{region '#Template'}
	{attribute 'Version' := '6.0.0.0'}
	{attribute 'Tags' := '"LCID": "1031", "Text": "AC, Aggregates, pre-heater"'}
	{attribute 'Tags' := '"LCID": "1033", "Text": "AC, Aggregates, pre-heater"'}
	{attribute 'Using' := '"Type": "Template", "URI": "Priority"'}		 
	{attribute 'Using' := '"Type": "Template", "URI": "BA2_Param"'}
	{attribute 'Using' := '"Type": "Template", "URI": "EC_ID"'}
	{attribute 'Description' := '"LCID": "1031", "Text": "Aggregat Vorerhitzer"'}
	{attribute 'Description' := '"LCID": "1033", "Text": "Aggregate pre-heater"'}
{endregion}
FUNCTION_BLOCK FB_BA_AC_PreHtr EXTENDS FB_BA_View
VAR_INPUT
	fSpTSuA					: REAL;
	fTSuA					: REAL;
	bSyncTSuACtrl			: BOOL;
	fSyncTSuACtrl			: REAL;	
	bDehumf					: BOOL;
	bSkipPreRinse			: BOOL; // Vorspülen überspringen // Skip pre-rinse
	fTWth					: REAL;
	bTWthLowLimit			: BOOL;
	bResetDehumf    		: BOOL;
END_VAR
VAR_OUTPUT
	bCmd					: BOOL;
	fPresentValue			: REAL;			
	bFrost					: BOOL;
	bPreRinseReady			: BOOL;  
	bActiveSeqCtrl			: BOOL;	
END_VAR
VAR_IN_OUT
	stTSeqLink				: ST_BA_SeqLink; // Sequenz Link Struktur // Sequence link structure	
	stAggregate				: ST_BA_Aggregate;	
END_VAR
VAR_INPUT CONSTANT PERSISTENT
	{attribute 'parameterCategory' := 'Behaviour'}
	fHysPuOn : REAL := 5.0;
	{attribute 'parameterCategory' := 'Behaviour'}
	fHysPuOff : REAL := 1.0;
END_VAR
VAR_INPUT CONSTANT
	TFl						: FB_BA_SensorAnalog;												
	TRt						: FB_BA_SensorAnalog;			
	TSuACtrl				: FB_BA_AC_PreHtrTSuACtrl;
	TRtCtrl					: FB_BA_AC_TRtCtrl;	
	TFrost					: FB_BA_SensorAnalog;																	
	TFrostPrtcCtrlAir		: FB_BA_PID_Sp;
	FrostThermostat			: FB_BA_SensorBinary;
	Vlv						: FB_BA_Vlv;
	Pu						: FB_BA_Pu1st;
	PlantLock				: FB_BA_PlantLock;			
	Aggregate				: FB_BA_Aggregate;																											 							
END_VAR
VAR
	bPrioSfty				: BOOL;
	bPrioCrit				: BOOL;		
	PrioSwiVal				: FB_BA_PrioSwi_B04;	
	
	HysPu					: FB_BA_Swi2P;
	SyncTSuACtrl			: FB_BA_RFTrig;
	SyncSeqCtrlIsActive		: FB_BA_RFTrig;
	PrioSwiSync				: FB_BA_PrioSwi_R04;	
END_VAR
VAR // added by the converter: edge detectors and wires of the graphical bodies
    _s1 : ST_BA_Analog;
    _s2 : ST_BA_Binary;
    _w1 : ANY;
    _w2 : BOOL;
END_VAR

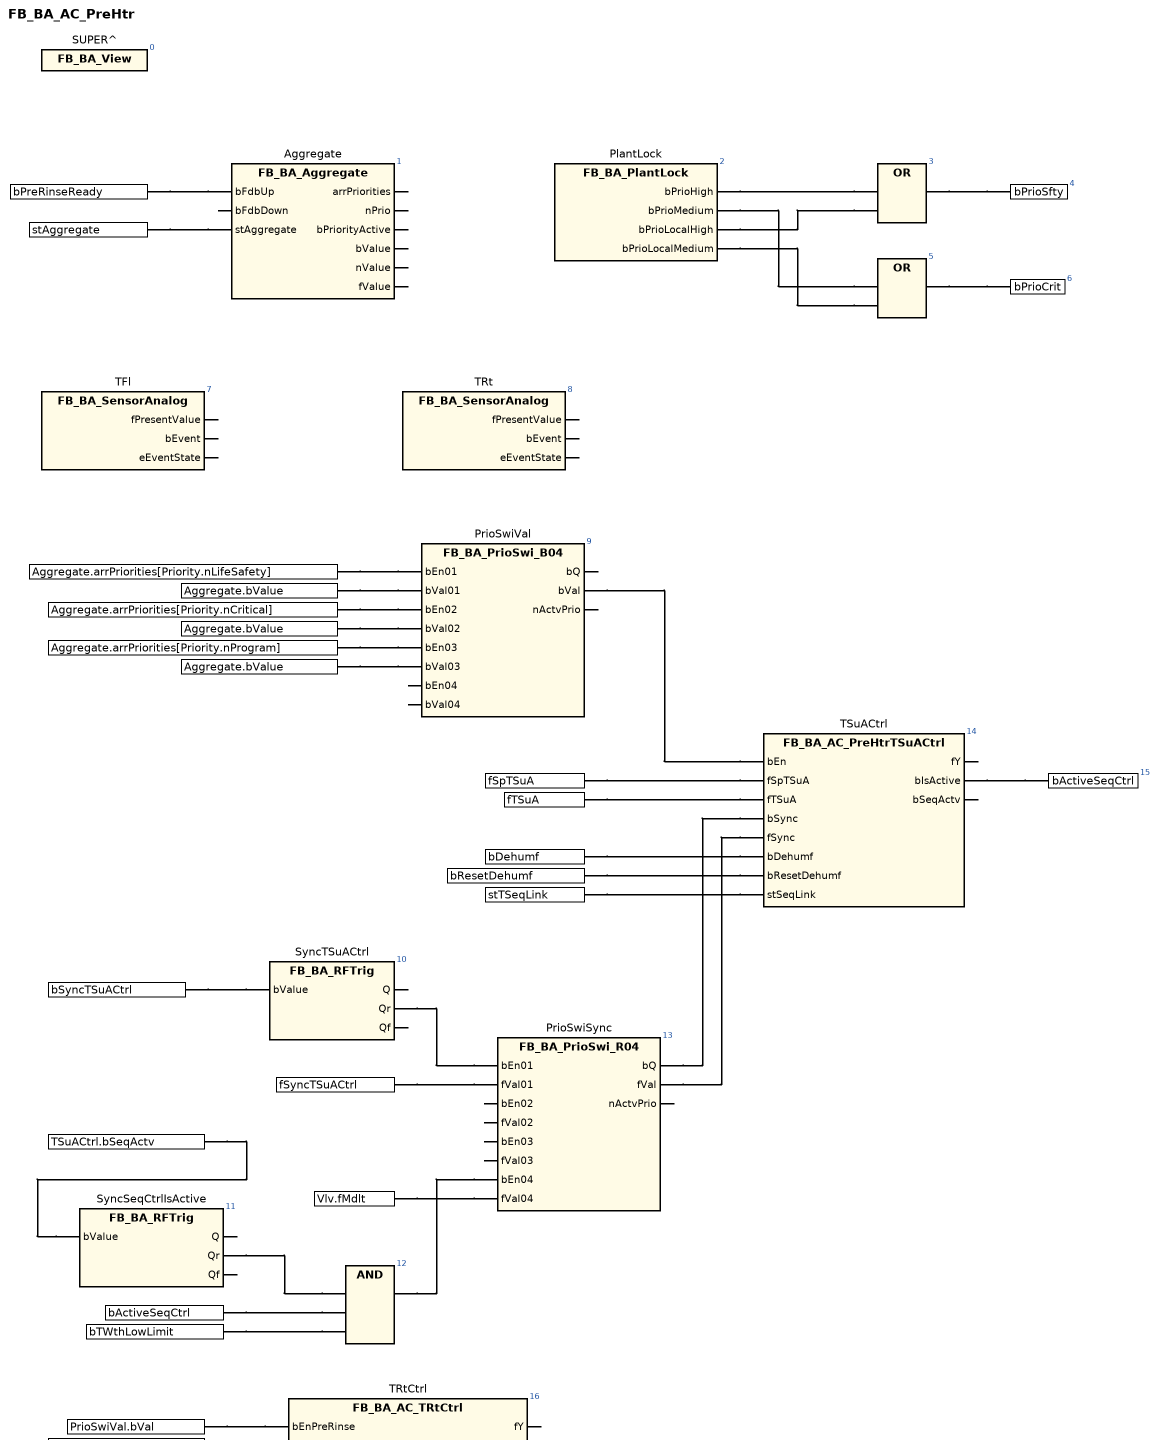
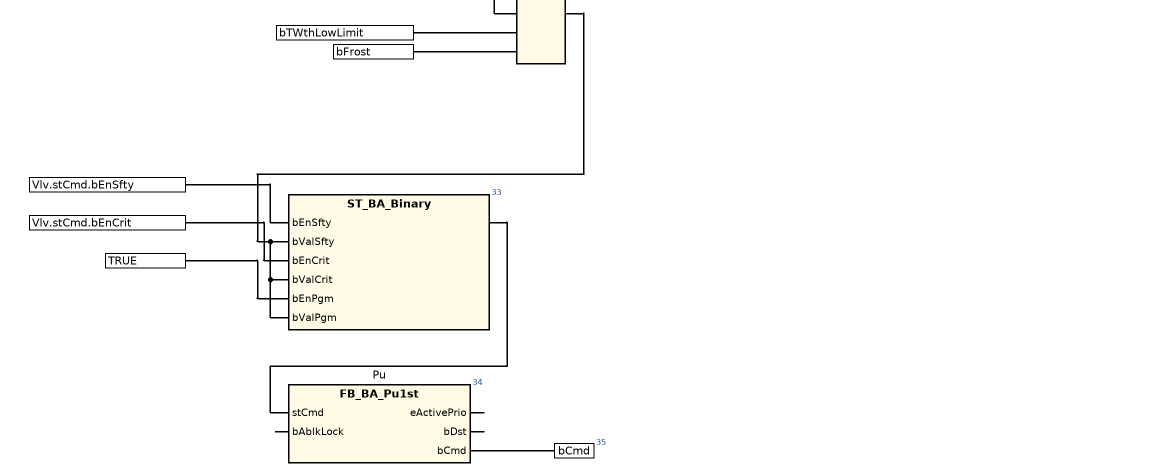
SUPER^(); // FB_BA_View
Aggregate(bFdbUp := bPreRinseReady, stAggregate := stAggregate); // FB_BA_Aggregate
PlantLock(); // FB_BA_PlantLock
bPrioSfty := PlantLock.bPrioHigh OR PlantLock.bPrioLocalHigh;
bPrioCrit := PlantLock.bPrioMedium OR PlantLock.bPrioLocalMedium;
TFl(); // FB_BA_SensorAnalog
TRt(); // FB_BA_SensorAnalog
PrioSwiVal(
    bEn01 := Aggregate.arrPriorities[Priority.nLifeSafety],
    bVal01 := Aggregate.bValue,
    bEn02 := Aggregate.arrPriorities[Priority.nCritical],
    bVal02 := Aggregate.bValue,
    bEn03 := Aggregate.arrPriorities[Priority.nProgram],
    bVal03 := Aggregate.bValue); // FB_BA_PrioSwi_B04
SyncTSuACtrl(bValue := bSyncTSuACtrl); // FB_BA_RFTrig
SyncSeqCtrlIsActive(bValue := TSuACtrl.bSeqActv); // FB_BA_RFTrig
PrioSwiSync(
    bEn01 := SyncTSuACtrl.Qr,
    fVal01 := fSyncTSuACtrl,
    bEn04 := SyncSeqCtrlIsActive.Qr AND bActiveSeqCtrl AND bTWthLowLimit,
    fVal04 := Vlv.fMdlt); // FB_BA_PrioSwi_R04
TSuACtrl(
    bEn := PrioSwiVal.bVal,
    fSpTSuA := fSpTSuA,
    fTSuA := fTSuA,
    bSync := PrioSwiSync.bQ,
    fSync := PrioSwiSync.fVal,
    bDehumf := bDehumf,
    bResetDehumf := bResetDehumf,
    stSeqLink := stTSeqLink); // FB_BA_AC_PreHtrTSuACtrl
bActiveSeqCtrl := TSuACtrl.bIsActive;
TRtCtrl(
    bEnPreRinse := PrioSwiVal.bVal,
    fTRt := TRt.fPresentValue,
    bTWthLowLimit := bTWthLowLimit,
    fTWth := fTWth,
    bSkipPreRinse := bSkipPreRinse,
    bSeqActive := stTSeqLink.bEnSeqLink); // FB_BA_AC_TRtCtrl
bPreRinseReady := TRtCtrl.bPreRinseReady;
TFrost(); // FB_BA_SensorAnalog
TFrostPrtcCtrlAir(bEn := TRUE, fX := TFrost.fPresentValue); // FB_BA_PID_Sp
FrostThermostat(); // FB_BA_SensorBinary
bFrost := TFrost.eEventState = E_BA_EventState.eLowLimit OR FrostThermostat.bPresentValue;
_w1 := MAX(TSuACtrl.fY, TRtCtrl.fY, TFrostPrtcCtrlAir.fY);
// compose _s1 : ST_BA_Analog
_s1.bEnSfty := Aggregate.arrPriorities[Priority.nLifeSafety] OR bPrioSfty;
_s1.fValSfty := _w1;
_s1.bEnCrit := Aggregate.arrPriorities[Priority.nCritical] OR bPrioCrit OR bFrost;
_s1.fValCrit := SEL(bFrost, _w1, 100);
_s1.bEnPgm := TRUE;
_s1.fValPgm := _w1;
Vlv(stCmd := _s1); // FB_BA_Vlv
fPresentValue := Vlv.fMdlt;
HysPu(bEn := TRUE, fIn := fPresentValue, fOn := fHysPuOn, fOff := fHysPuOff); // FB_BA_Swi2P
_w2 := HysPu.bQ OR bTWthLowLimit OR bFrost;
// compose _s2 : ST_BA_Binary
_s2.bEnSfty := Vlv.stCmd.bEnSfty;
_s2.bValSfty := _w2;
_s2.bEnCrit := Vlv.stCmd.bEnCrit;
_s2.bValCrit := _w2;
_s2.bEnPgm := TRUE;
_s2.bValPgm := _w2;
Pu(stCmd := _s2); // FB_BA_Pu1st
bCmd := Pu.bCmd;

METHOD FB_init : BOOL
VAR_INPUT
	bInitRetains : BOOL; // if TRUE, the retain variables are initialized (warm start / cold start)
	bInCopyCode : BOOL;  // if TRUE, the instance afterwards gets moved into the copy code (online change)
END_VAR
PlantLock.Parent								:= THIS^;		

TFl.iParent										:= THIS^;		
TFl.iLabel										:= LblAgg_TemperatureFlow;   
TFl.sObjectName									:= '{Idx=11}';						 
TFl.eDPADMode									:= E_BA_DPADMode.eInclude;
TFl.MV.eUnit									:= E_BA_Unit.eTemperature_DegreesCelsius;
TFl.MV.fResolution 								:= 0.01;
TFl.MV.fScaleOffset 							:= 0; 
TFl.MV.bEventDetectionEnable					:= TRUE;
TFl.MV.eEnPlantLock								:= E_BA_LockPriority.eNoLock;
                            					                            					
TRt.iParent										:= THIS^;		
TRt.iLabel										:= LblAgg_TemperatureReturnFlow;   
TRt.sObjectName									:= '{Idx=11}';						 
TRt.eDPADMode									:= E_BA_DPADMode.eInclude;
TRt.MV.eUnit									:= E_BA_Unit.eTemperature_DegreesCelsius;
TRt.MV.fResolution 								:= 0.01;
TRt.MV.fScaleOffset 							:= 0;  
TRt.MV.bEventDetectionEnable					:= TRUE;
TRt.MV.eEnPlantLock								:= E_BA_LockPriority.eMedium;

TSuACtrl.iParent								:= THIS^;	
TSuACtrl.iLabel									:= LblCtl_SupplyAirTemperatureControl;   
TSuACtrl.sObjectName							:= '{Idx=11}';						 
TSuACtrl.eDPADMode								:= E_BA_DPADMode.eInclude;								

TRtCtrl.iParent									:= THIS^;
TRtCtrl.iLabel									:= LblCtl_ReturnWaterControl;   
TRtCtrl.sObjectName								:= '{Idx=12}';						 
TRtCtrl.eDPADMode								:= E_BA_DPADMode.eInclude;								
TRtCtrl.PreRinseDst.bEventDetectionEnable		:= TRUE;
TRtCtrl.PreRinseDst.eEnPlantLock				:= E_BA_LockPriority.eNoLock;
	                                				
TFrost.iParent									:= THIS^;		
TFrost.iLabel									:= LblCtl_TemperatureFrost;   
TFrost.sObjectName								:= '{Idx=11}';						 
TFrost.eDPADMode								:= E_BA_DPADMode.eInclude;
TFrost.MV.eUnit									:= E_BA_Unit.eTemperature_DegreesCelsius;
TFrost.MV.fResolution 							:= 0.0004577776;
TFrost.MV.fScaleOffset 							:= 0;  
TFrost.MV.bEventDetectionEnable					:= TRUE;
TFrost.MV.eEnPlantLock							:= E_BA_LockPriority.eMedium;

TFrostPrtcCtrlAir.iParent						:= THIS^;	
TFrostPrtcCtrlAir.iLabel						:= LblCtl_FrostProtectionControl;   
TFrostPrtcCtrlAir.sObjectName					:= '{Idx=13}';						 
TFrostPrtcCtrlAir.eDPADMode						:= E_BA_DPADMode.eInclude;
TFrostPrtcCtrlAir.Sp.fValueRm 					:= 5.0;
TFrostPrtcCtrlAir.Ctrl.fProportionalConstant	:= 5;
TFrostPrtcCtrlAir.Ctrl.fIntegralConstant		:= 60;	
TFrostPrtcCtrlAir.Ctrl.eActionRm				:= E_BA_Action.eReverse;

FrostThermostat.iParent							:= THIS^; 
FrostThermostat.iLabel							:= LblAgg_FrostProtectionMonitor;   
FrostThermostat.sObjectName						:= '{Idx=13}';						 
FrostThermostat.eDPADMode						:= E_BA_DPADMode.eInclude;
FrostThermostat.Input.iLabel					:= LblFun_OperationalMessage;   
FrostThermostat.Input.sObjectName				:= '{Idx=13}';						 
FrostThermostat.Input.ePolarity					:= E_BA_Polarity.eReverse;
FrostThermostat.Input.sActiveText 				:= txtEvent_Triggered;
FrostThermostat.Input.sInactiveText 			:= txtEvent_Normal;
FrostThermostat.Input.nEventClassID				:= EC_ID.NC30;
FrostThermostat.Input.aEventTransitionText[1]	:= txtEvent_Triggered;
FrostThermostat.Input.aEventTransitionText[2]	:= txtEvent_Error;
FrostThermostat.Input.aEventTransitionText[3]	:= txtEvent_Normal;
FrostThermostat.Input.bEventDetectionEnable		:= TRUE;
FrostThermostat.Input.eEnPlantLock				:= E_BA_LockPriority.eMedium;	

Vlv.iParent										:= THIS^;
Vlv.iLabel										:= LblAgg_Valve;    									 
Vlv.sObjectName									:= '{Idx=11}';						 
Vlv.eDPADMode									:= E_BA_DPADMode.eInclude;								
                            					
Pu.iParent										:= THIS^;
Pu.iLabel										:= LblAgg_Pump;   									 
Pu.sObjectName									:= '{Idx=11}';						 
Pu.eDPADMode									:= E_BA_DPADMode.eInclude;
Pu.Dst.bEventDetectionEnable					:= TRUE;
Pu.Dst.eEnPlantLock								:= E_BA_LockPriority.eMedium;
END_METHOD

END_FUNCTION_BLOCK

(* stored: Version 1.1.0.1, ProductVersion 3.1.4024.12
   POU FB_BA_AC_PreHtr: Id {5ffe416f-f0a8-4ab4-9678-c819530d6896}, SpecialFunc None
   Method FB_init: Id {29b5dac5-ce3e-49b5-bfbd-f6a3d8a17392} *)
